FUNCTION_BLOCK InvokingTasks EXTENDS TcoCore.TcoContext
VAR
	Cylinder : TcoPneumatics.fbCylinder(THIS^);
	
	TriggerHome : BOOL;
	TriggerWork : BOOL;


	
	//simulate IO
	AtHome:BOOL;
	AtWork:BOOL;
	ToHome:BOOL;
	ToWork:BOOL;
	
	_simTimerValue : UINT := 500;
	_simTimer : Tc2_Standard.TON;

END_VAR

//Use main method

(*~
	<docu>
		<summary>
			Main method of the TcoContext. This is the entry point of any control logic that belongs to this context. 
			The call of this method is ensured by calling the <c>InstanceName.Run()</c> method, and it must not be called explicitly.
			This method is abstract, and it must be overridden in derived block.
		</summary>
	</docu>
~*)
METHOD PROTECTED  Main
VAR_INST
	ToHomeTemp:BOOL;
	ToWorkTemp:BOOL;

END_VAR
Cylinder
(
	inAtHomePos := AtHome,
	inAtWorkPos := AtWork,
	outToHomePos => ToHome,
	outToWorkPos => ToWork
);

IF ToWork THEN
	AtHome := FALSE;
	_simTimer(IN:=TRUE,PT:= UINT_TO_TIME(_simTimerValue*4));
	IF(_simTimer.Q) THEN
		AtWork :=TRUE;
		_simTimer(IN:=FALSE,PT:= UINT_TO_TIME(0));
		Cylinder.Restore();
	END_IF
END_IF


IF ToHome THEN
	AtWork := FALSE;
	_simTimer(IN:=TRUE,PT:= UINT_TO_TIME(_simTimerValue*4));
	IF(_simTimer.Q) THEN
		AtHome :=TRUE;
		_simTimer(IN:=FALSE,PT:= UINT_TO_TIME(0));
		Cylinder.Restore();
	END_IF
END_IF

Cylinder.Service(); //enable manual control
END_METHOD

END_FUNCTION_BLOCK

(* stored: Version 1.1.0.1, ProductVersion 3.1.4024.6
   POU InvokingTasks: Id {12cfae65-b95f-0775-1a26-802c03070a44}, SpecialFunc None
   Method Main: Id {a6ba057b-ec5a-0051-11a4-7a811a9c8902} *)
